FUNCTION_BLOCK Json
VAR_INPUT
END_VAR
VAR_OUTPUT
	payload: STRING(255);
END_VAR
VAR
  writer: FB_JsonSaxWriter;
END_VAR

METHOD create : STRING(255)
VAR_INPUT
	fromString: STRING(255);
END_VAR
writer.StartObject();
writer.AddKey('message');
writer.AddString(fromString);
writer.EndObject();
payload := writer.GetDocument();
writer.ResetDocument();
create := payload;
END_METHOD

END_FUNCTION_BLOCK

(* stored: Version 1.1.0.1, ProductVersion 3.1.4024.12
   POU Json: Id {c50ea90b-f9f2-4eba-85a8-23aaa103e8e0}, SpecialFunc None
   Method create: Id {595df800-60b9-4f40-bb41-6806137d1ad6} *)
